FUNCTION_BLOCK FB_ConveyorControl
(*
Version history:
DATE		|	Version/Author 		|	Remark
----------------------------------------------------------------------------------------------------
16.03.12	|	2.000.001	PSA		|	Original Version.
									|	Runs a given Conveyor.
									|	Generic block to run any conveyor.
*)
VAR_INPUT
	bEnableConveyor      			: BOOL;				(* Enable this conveyor *)
	bPhysicalMotorOK				: BOOL;				(* Drive is OK *)
	bMachineIsReset					: BOOL;				(* Reset *)
	bConveyorStart					: BOOL;				(* Conveyor start requested *)
	bConveyorStop					: BOOL;				(* Conveyor stop requested *)
	bConveyorTimeOut				: BOOL;				(* PreMachine is running *)
	nConveyorRunSpeed				: WORD;				(* Set speed for the conveyor *)
	nScalingFactor					: WORD;				(* Scaling factor for the conveyor output *)
	fConveyorStopsAfterTimeSet		: LREAL;			(* Maximum conveyor run time *)
END_VAR
VAR_OUTPUT
	bConveyorRunLamp				: BOOL;
	bConveyorEnabled				: BOOL;
	bConveyorRun					: BOOL;
	bConStopTimeOut					: BOOL;
	nConveyorAnalogueOutputSpeed	: INT;
END_VAR
VAR
	bFlashOut						: BOOL;
	fbConveyorStopTimer				: TON;
	fbBlink1						: FB_Blink;
END_VAR

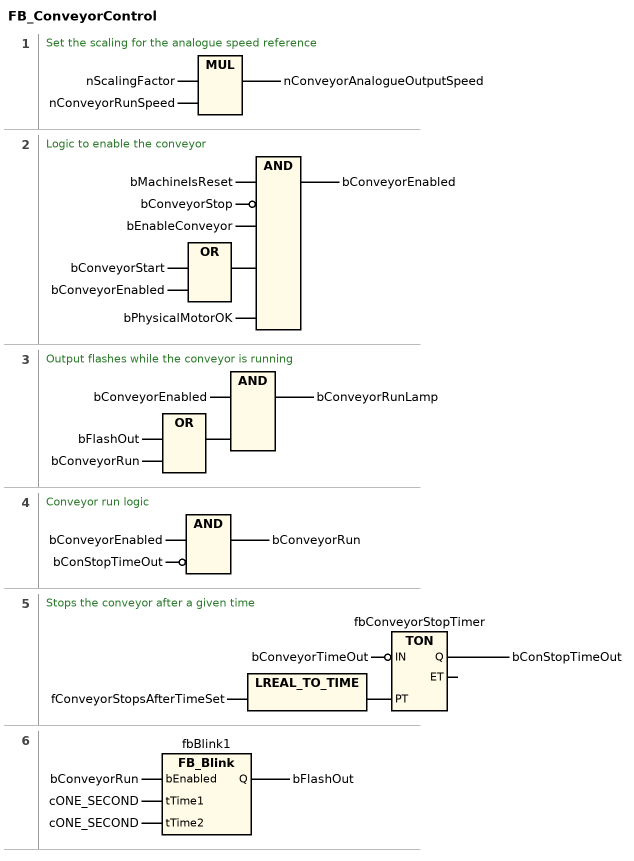
// NETWORK 1
// Set the scaling for the analogue speed reference
nConveyorAnalogueOutputSpeed := nScalingFactor * nConveyorRunSpeed;

// NETWORK 2
// Logic to enable the conveyor
bConveyorEnabled := bMachineIsReset AND NOT bConveyorStop AND bEnableConveyor AND (bConveyorStart OR bConveyorEnabled) AND bPhysicalMotorOK;

// NETWORK 3
// Output flashes while the conveyor is running
bConveyorRunLamp := bConveyorEnabled AND (bFlashOut OR bConveyorRun);

// NETWORK 4
// Conveyor run logic
bConveyorRun := bConveyorEnabled AND NOT bConStopTimeOut;

// NETWORK 5
// Stops the conveyor after a given time
fbConveyorStopTimer(IN := NOT bConveyorTimeOut, PT := LREAL_TO_TIME(fConveyorStopsAfterTimeSet)); // TON
bConStopTimeOut := fbConveyorStopTimer.Q;

// NETWORK 6
fbBlink1(bEnabled := bConveyorRun, tTime1 := cONE_SECOND, tTime2 := cONE_SECOND); // FB_Blink
bFlashOut := fbBlink1.Q;

END_FUNCTION_BLOCK

(* stored: Version 1.1.0.1, ProductVersion 3.1.4024.15
   POU FB_ConveyorControl: Id {c30ccc34-a939-4511-99f0-a5133a8a282f}, SpecialFunc None *)
